TYPE "UDT_Device_HMI"
VERSION : 0.1
   STRUCT
      IN_xManualStart : Bool;   //    手动启动
      IN_xManualStop : Bool;   //    手动停止
      OUT_uiState : UInt;   //    状态字(0=初始状态,1=已停止,2=已启动,3=正在启动,4=正在停止,5=停止故障,6=启动故障,7=设备报警)
   END_STRUCT;

END_TYPE